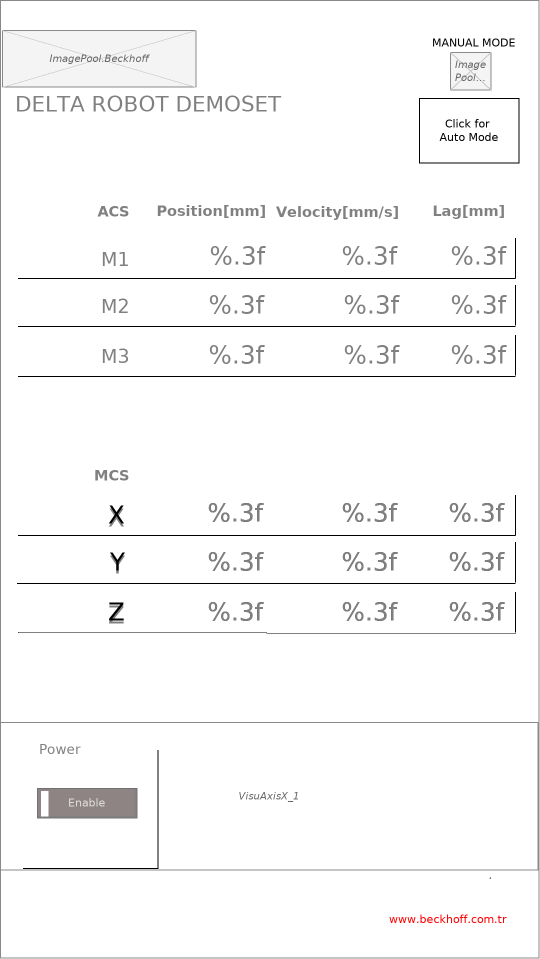
VISUALIZATION Visualization_AxesInfo_Manual  // 540x959, background image ImagePool.Background
    Textfield (8,590 120x50), "Z", invisible if: GVL_Process.bManualSelectZ
    Textfield (8,540 120x50), "Y", invisible if: GVL_Process.bManualSelectY
    Textfield (8,493 120x50), "X", invisible if: GVL_Process.bManualSelectX
    Textfield (8,537 120x50), "Y", invisible if: not GVL_Process.bManualSelectY
        p2073431371: GVL_Process.nSizeSelectY
    Frame (0,722 538x148)
        shows VisuAxisX_1()
        shows VisuAxisY_1()
        shows VisuAxisZ_1()
    Label (12,77 308x54), "DELTA ROBOT DEMOSET"
    Label (35,229 155x61), "M1"
    Textfield (148,231 120x50), "%.3f", text variable: GVL_Axis.AxisM1_B.NcToPlc.ActPos
    Rectangle (39,248 7x22), invisible if: not stAxisM1_B.Out.xEnabled
    Rectangle (27,248 7x22), invisible if: not stAxisM1_B.Out.xAxisError
    Label (11,183 122x57), "ACS"
    Label (149,186 120x50), "Position[mm]"
    Label (276,187 126x50), "Velocity[mm/s]"
    Textfield (280,231 120x50), "%.3f", text variable: GVL_Axis.AxisM1_B.NcToPlc.ActVelo
    Image (2,30 194x57), image: ImagePool.Beckhoff
    Label (388,186 120x50), "Lag[mm]"
    Textfield (389,231 120x50), "%.3f", text variable: GVL_Axis.AxisM1_B.NcToPlc.PosDiff
    Line (18,278) (515,278)
    Line (515,238) (515,278)
    Label (38,276 155x61), "M2"
    Textfield (147,280 120x50), "%.3f", text variable: GVL_Axis.AxisM2_C.NcToPlc.ActPos
    Rectangle (39,295 7x22), invisible if: not stAxisM2_C.Out.xEnabled
    Rectangle (27,295 7x22), invisible if: not stAxisM2_C.Out.xAxisError
    Textfield (282,280 120x50), "%.3f", text variable: GVL_Axis.AxisM2_C.NcToPlc.ActVelo
    Textfield (389,280 120x50), "%.3f", text variable: GVL_Axis.AxisM2_C.NcToPlc.PosDiff
    Line (515,285) (515,325)
    Label (38,326 155x61), "M3"
    Textfield (147,330 120x50), "%.3f", text variable: GVL_Axis.AxisM3_A.NcToPlc.ActPos
    Rectangle (39,345 7x22), invisible if: not stAxisM3_A.Out.xEnabled
    Rectangle (27,345 7x22), invisible if: not stAxisM3_A.Out.xAxisError
    Textfield (282,330 120x50), "%.3f", text variable: GVL_Axis.AxisM3_A.NcToPlc.ActVelo
    Textfield (389,330 120x50), "%.3f", text variable: GVL_Axis.AxisM3_A.NcToPlc.PosDiff
    Line (18,376) (515,376)
    Line (515,335) (515,375)
    Line (18,326) (515,326)
    Label (11,447 122x57), "MCS"
    Textfield (126,488 140x50), "%.3f", text variable: GVL_Axis.AxisX.NcToPlc.ActPos, invisible if: not GVL_Process.bManualSelectX
        p2073431371: GVL_Process.nSizeSelectX
    Rectangle (39,505 7x22), invisible if: not stAxisX.Out.xEnabled
    Rectangle (27,505 7x22), invisible if: not stAxisX.Out.xAxisError
    Textfield (280,488 120x50), "%.3f", text variable: GVL_Axis.AxisX.NcToPlc.ActVelo, invisible if: not GVL_Process.bManualSelectX
        p2073431371: GVL_Process.nSizeSelectX
    Textfield (387,488 120x50), "%.3f", text variable: GVL_Axis.AxisX.NcToPlc.PosDiff, invisible if: not GVL_Process.bManualSelectX
        p2073431371: GVL_Process.nSizeSelectX
    Line (18,535) (515,535), colour toggle: GVL_Process.bManualSelectX
    Line (515,495) (515,535), colour toggle: GVL_Process.bManualSelectX
    Textfield (126,537 140x50), "%.3f", text variable: GVL_Axis.AxisY.NcToPlc.ActPos, invisible if: not GVL_Process.bManualSelectY
        p2073431371: GVL_Process.nSizeSelectY
    Rectangle (39,552 7x22), invisible if: not stAxisY.Out.xEnabled
    Rectangle (27,552 7x22), invisible if: not stAxisY.Out.xAxisError
    Textfield (280,537 120x50), "%.3f", text variable: GVL_Axis.AxisY.NcToPlc.ActVelo, invisible if: not GVL_Process.bManualSelectY
        p2073431371: GVL_Process.nSizeSelectY
    Textfield (387,537 120x50), "%.3f", text variable: GVL_Axis.AxisY.NcToPlc.PosDiff, invisible if: not GVL_Process.bManualSelectY
        p2073431371: GVL_Process.nSizeSelectY
    Line (515,542) (515,582), colour toggle: GVL_Process.bManualSelectY
    Textfield (126,587 140x50), "%.3f", text variable: GVL_Axis.AxisZ.NcToPlc.ActPos, invisible if: not GVL_Process.bManualSelectZ
        p2073431371: GVL_Process.nSizeSelectZ
    Rectangle (39,602 7x22), invisible if: not stAxisZ.Out.xEnabled
    Rectangle (27,602 7x22), invisible if: not stAxisZ.Out.xAxisError
    Textfield (280,587 120x50), "%.3f", text variable: GVL_Axis.AxisZ.NcToPlc.ActVelo, invisible if: not GVL_Process.bManualSelectZ
        p2073431371: GVL_Process.nSizeSelectZ
    Textfield (387,587 120x50), "%.3f", text variable: GVL_Axis.AxisZ.NcToPlc.PosDiff, invisible if: not GVL_Process.bManualSelectZ
        p2073431371: GVL_Process.nSizeSelectZ
    Line (18,632) (515,633), colour toggle: GVL_Process.bManualSelectZ
    Line (515,592) (515,632), colour toggle: GVL_Process.bManualSelectZ
    Line (17,583) (515,583), colour toggle: GVL_Process.bManualSelectY
    Textfield (8,490 120x50), "X", invisible if: not GVL_Process.bManualSelectX
        p2073431371: GVL_Process.nSizeSelectX
    Textfield (8,587 120x50), "Z", invisible if: not GVL_Process.bManualSelectZ
        p2073431371: GVL_Process.nSizeSelectZ
    Textfield (126,537 140x50), "%.3f", text variable: GVL_Axis.AxisY.NcToPlc.ActPos, invisible if: GVL_Process.bManualSelectY
    Textfield (280,537 120x50), "%.3f", text variable: GVL_Axis.AxisY.NcToPlc.ActVelo, invisible if: GVL_Process.bManualSelectY
    Textfield (387,537 120x50), "%.3f", text variable: GVL_Axis.AxisY.NcToPlc.PosDiff, invisible if: GVL_Process.bManualSelectY
    Textfield (126,488 140x50), "%.3f", text variable: GVL_Axis.AxisX.NcToPlc.ActPos, invisible if: GVL_Process.bManualSelectX
    Textfield (280,488 120x50), "%.3f", text variable: GVL_Axis.AxisX.NcToPlc.ActVelo, invisible if: GVL_Process.bManualSelectX
    Textfield (387,488 120x50), "%.3f", text variable: GVL_Axis.AxisX.NcToPlc.PosDiff, invisible if: GVL_Process.bManualSelectX
    Textfield (126,587 140x50), "%.3f", text variable: GVL_Axis.AxisZ.NcToPlc.ActPos, invisible if: GVL_Process.bManualSelectZ
    Textfield (280,587 120x50), "%.3f", text variable: GVL_Axis.AxisZ.NcToPlc.ActVelo, invisible if: GVL_Process.bManualSelectZ
    Textfield (387,587 120x50), "%.3f", text variable: GVL_Axis.AxisZ.NcToPlc.PosDiff, invisible if: GVL_Process.bManualSelectZ
    Label (373,882 150x75), "www.beckhoff.com.tr"
    Group (23,721 136x148)
        Button (14,67 100x30), "Enable"
            toggle GVL_Process.bAllAxesEnable
        Rectangle (18,70 7x25), invisible if: not GVL_Process.bAllAxesEnable
        Line (0,147) (135,147)
        Line (135,147) (135,29)
        Label (2,0 70x57), "Power"
    InvisibleInput (8,485 510x51), input disabled if: GVL_Process.bManualSelectX
        toggle GVL_Process.bManualSelectX
        OnMouseClick: FrameSelectionChange Selection=SelectedFrame=4ba14cc2-2c84-48fd-8925-52c85ec640bd, GlobSel=AssignType=Directly, SelType=Locally
    InvisibleInput (8,585 510x51), input disabled if: GVL_Process.bManualSelectZ
        toggle GVL_Process.bManualSelectZ
        OnMouseClick: FrameSelectionChange Selection=SelectedFrame=4ba14cc2-2c84-48fd-8925-52c85ec640bd, Selection=2, GlobSel=AssignType=Directly, SelType=Locally
    InvisibleInput (8,535 510x51), input disabled if: GVL_Process.bManualSelectY
        toggle GVL_Process.bManualSelectY
        OnMouseClick: FrameSelectionChange Selection=SelectedFrame=4ba14cc2-2c84-48fd-8925-52c85ec640bd, Selection=1, GlobSel=AssignType=Directly, SelType=Locally
    Image (450,52 41x38), image: ImagePool.Mode_icon
        OnMouseMove: execute { GVL_Process.bMessageBubbleMan:=TRUE; }
        OnMouseClick: change screen: Visualization_AxesInfo
        OnMouseLeave: execute { GVL_Process.bMessageBubbleMan := FALSE; }
    Label (424,29 100x28), "MANUAL MODE"
    Rectangle (419,98 100x65), "Click for Auto Mode", invisible if: not GVL_Process.bMessageBubbleMan
    Rectangle (490,877 0x1)
END_VISUALIZATION

(* stored: Version 1.1.0.1, ProductVersion 3.1.4022.6
   Visu Visualization_AxesInfo_Manual: Id {ff9fe4be-b2e1-4450-87a0-26816c4c141a} *)
